FUNCTION_BLOCK sql_parameters IMPLEMENTS InterfaceSQLParameters
VAR_INPUT
END_VAR
VAR_OUTPUT
END_VAR
VAR
	_parameter : ARRAY [1..DbLibParam.MAX_COLUMN_NUM] OF ST_ExpParameter;
	_table_name : T_MaxString;
	_p_data : PVOID;
	_cb_data : UDINT;
END_VAR
VAR PERSISTENT
	current_column_index : UDINT := 0;
END_VAR

{warning 'add method implementation '}
METHOD add_column : BOOL
VAR_INPUT
	sParaName : T_MaxString;
	eParaType : E_ExpParameterType;
	nParaSize : UDINT;
END_VAR
IF DbLibParam.MAX_COLUMN_NUM <= current_column_index THEN
	add_column := FALSE;
	RETURN;
END_IF 
current_column_index := current_column_index + 1;
_parameter[current_column_index].sParaName := sParaName;
_parameter[current_column_index].eParaType := eParaType;
_parameter[current_column_index].nParaSize := nParaSize;
add_column := TRUE;
END_METHOD

{warning 'add property implementation'}
PROPERTY cbData : UDINT
GET
cbData := _cb_data;
END_GET
SET
_cb_data := cbData;
END_SET
END_PROPERTY

{warning 'add property implementation'}
PROPERTY cbParameters : UDINT
GET
IF current_column_index = 0 THEN
	cbParameters := 0;
ELSE
	cbParameters := SIZEOF(_parameter[1]) * current_column_index;
END_IF
END_GET
END_PROPERTY

{warning 'add property implementation'}
PROPERTY column_num : UDINT
GET
column_num := current_column_index;
END_GET
END_PROPERTY

{warning 'add property implementation'}
PROPERTY insert_query_string : Tc2_System.T_MaxString
GET
VAR
	i : UDINT;
END_VAR
insert_query_string := 'INSERT INTO (';
FOR i := 1 TO current_column_index DO
	IF i > 1 THEN
		insert_query_string := CONCAT(insert_query_string,', ');	
	END_IF
	insert_query_string := CONCAT(insert_query_string,_parameter[i].sParaName);
END_FOR
insert_query_string := CONCAT(insert_query_string, ') VALUES (');
FOR i := 1 TO current_column_index DO
	IF i > 1 THEN
		insert_query_string := CONCAT(insert_query_string,', ');
	END_IF
	insert_query_string := CONCAT(insert_query_string,'{');
	insert_query_string := CONCAT(insert_query_string,_parameter[i].sParaName);
	insert_query_string := CONCAT(insert_query_string,'}');
END_FOR
insert_query_string := CONCAT(insert_query_string, ')');
END_GET
END_PROPERTY

{warning 'add property implementation'}
PROPERTY pData : PVOID
GET
pData := _p_data;
END_GET
SET
_p_data := pData;
END_SET
END_PROPERTY

{warning 'add property implementation'}
PROPERTY pParameters : PVOID
GET
pParameters := ADR(_parameter[1]);
END_GET
END_PROPERTY

{warning 'add property implementation'}
PROPERTY table_name : Tc2_System.T_MaxString
GET
table_name := _table_name;
END_GET
SET
_table_name := table_name;
END_SET
END_PROPERTY

END_FUNCTION_BLOCK

(* stored: Version 1.1.0.1, ProductVersion 3.1.4024.12
   POU sql_parameters: Id {733fc625-5004-4381-879d-5fd7fccfb98f}, SpecialFunc None
   Method add_column: Id {3b73a0cd-b383-44c6-a93e-cf5898849a7a}
   Property cbData: Id {b17533ce-5c5e-4d02-8687-221f6a6deaa5}
   Get Get: Id {55720e52-3e48-4e81-9fcb-fd354efa472a}
   Set Set: Id {7a4034be-c45d-4e8c-a129-31a067bb62d7}
   Property cbParameters: Id {6ec10b35-7838-4ddb-a63f-45a5ed1677e7}
   Get Get: Id {7e3b93c9-7202-4872-b722-392873fe6049}
   Property column_num: Id {a64ad4a4-be4f-43db-b542-33e773d74a7f}
   Get Get: Id {cff8c15a-81b2-4296-a657-71990fd63ecd}
   Property insert_query_string: Id {e09d6d70-0c52-455b-ac7b-cf616cbdfa61}
   Get Get: Id {8b0c9427-cca9-4494-af85-d8b8e32748b2}
   Property pData: Id {c3313b35-5ea9-4b65-8028-8f7ae4095e68}
   Get Get: Id {9a654a41-ee0a-4c0f-a77d-c77606019674}
   Set Set: Id {4c3a6f50-5687-4ae8-a106-e397b5b3b534}
   Property pParameters: Id {dd20c012-0a16-4b1b-b2e9-16cd13f4d32a}
   Get Get: Id {ff466214-aa18-493c-bad6-022db1cbd49c}
   Property table_name: Id {e38de48c-6b0f-45b6-8fa4-67575a9cf6f9}
   Get Get: Id {f85e7fa5-a341-4565-982c-4e4bcc4b1ec2}
   Set Set: Id {6d1eb162-e420-460a-a5da-2d2fd4bb40c2} *)
